FUNCTION_BLOCK FB_GamePlay
VAR_INPUT
END_VAR
VAR_OUTPUT
END_VAR
VAR
END_VAR

// Decode sequencer step bits
MEMSET(ADR(GVL_Global.bStep), 0, SIZEOF(GVL_Global.bStep));
GVL_Global.bStep[GVL_Global.iStepNumber] := TRUE;

//States
// 0 = Idle - Game is waiting for user to start game
IF GVL_Global.bStep[0] THEN
	IF GVL_Global.stGamePlay.bClear THEN
		GVL_Global.iStepNumber := 1;
	END_IF
	
	IF GVL_Global.stGamePlay.bStart THEN
		GVL_Global.iStepNumber := 2;
	END_IF
	
// 1 = Clear - Clear all variables
ELSIF GVL_Global.bStep[1] THEN
	FB_Clear();
	IF GVL_Global.bClear_Complete THEN
		GVL_Global.stGamePlay.bClear := FALSE;
		GVL_Global.bClear_Complete := FALSE;
		GVL_Global.iStepNumber := 0;
	END_IF
	
// 2 = Game Set Up - Game to get set up to play
ELSIF GVL_Global.bStep[2] THEN
	IF GVL_Global.bReadyToStart THEN
		IF GVL_Global.bInitialStart THEN
			FB_GameSetup();
			IF GVL_Global.stGameSetup.bGameSetupComplete THEN
				GVL_Global.bInitialStart := FALSE;
				GVL_Global.bGameInProgress := TRUE;
				GVL_Global.iStepNumber := 3;
			END_IF
		ELSE
			IF GVL_Global.bGameInProgress THEN
				GVL_Global.iStepNumber := 3;
			ELSE
				GVL_Global.iStepNumber := 0;
			END_IF
		END_IF
	ELSE
		FB_Clear();
	END_IF
	
// 3 = Game Is Ongoing - Game is currently being played
ELSIF GVL_Global.bStep[3] THEN
	IF GVL_Global.bGameInProgress THEN
		;
	END_IF
	;
	
// 4 = Pause Game - Game is paused or people have left the table
ELSIF GVL_Global.bStep[4] THEN
	;
	
// 5 = End Game - Finish game and display results
ELSIF GVL_Global.bStep[5] THEN
	;
// 63-999 = Error State
ELSIF GVL_Global.bStep[63] THEN
	;
END_IF

END_FUNCTION_BLOCK

(* stored: Version 1.1.0.1, ProductVersion 3.1.4024.10
   POU FB_GamePlay: Id {6b6e1877-5bf4-42b4-a300-e43fe1977a81}, SpecialFunc None *)
